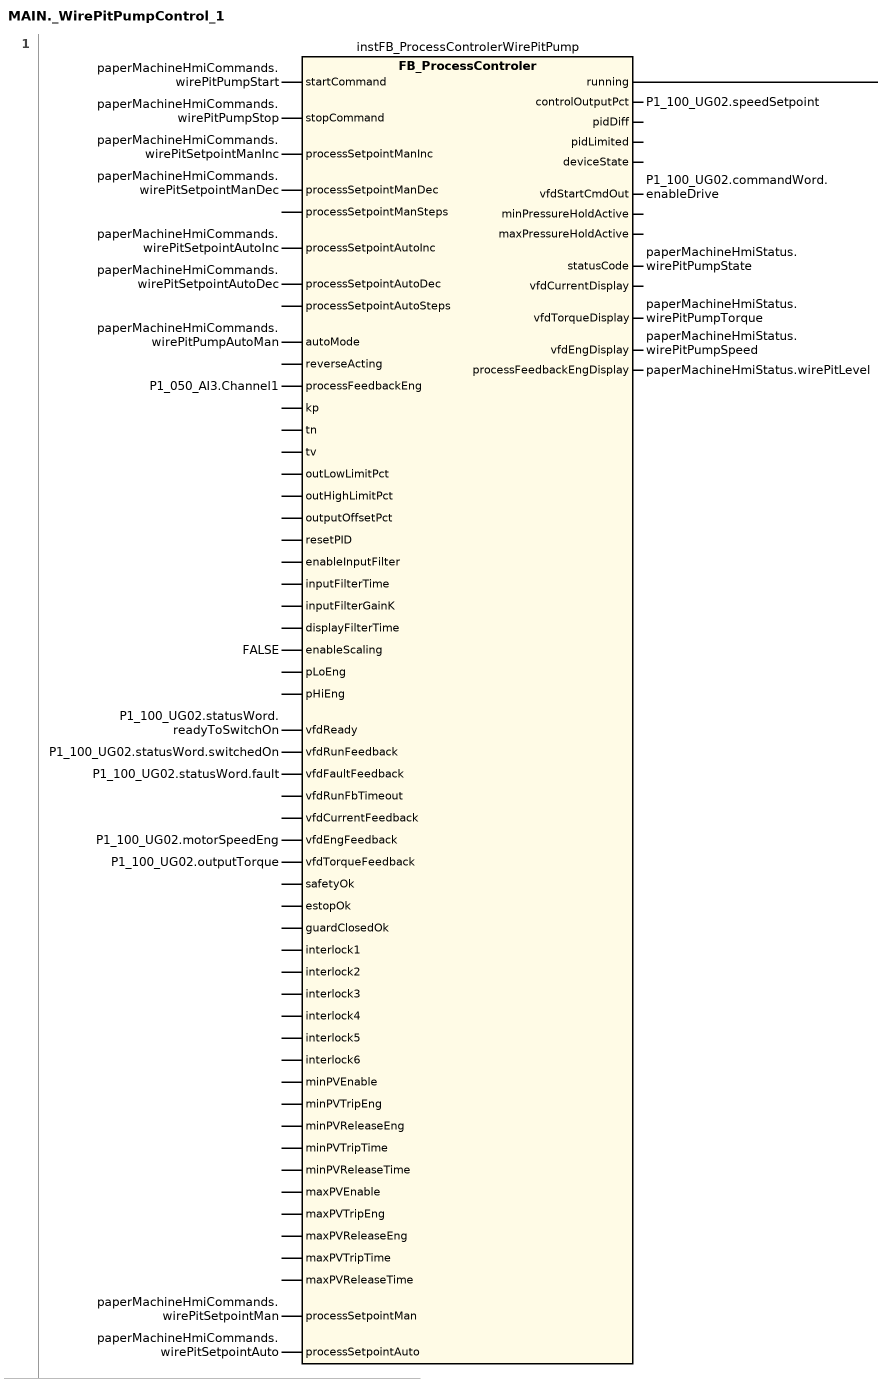
// NETWORK 1
instFB_ProcessControlerWirePitPump(
    startCommand := paperMachineHmiCommands.wirePitPumpStart,
    stopCommand := paperMachineHmiCommands.wirePitPumpStop,
    processSetpointManInc := paperMachineHmiCommands.wirePitSetpointManInc,
    processSetpointManDec := paperMachineHmiCommands.wirePitSetpointManDec,
    processSetpointAutoInc := paperMachineHmiCommands.wirePitSetpointAutoInc,
    processSetpointAutoDec := paperMachineHmiCommands.wirePitSetpointAutoDec,
    autoMode := paperMachineHmiCommands.wirePitPumpAutoMan,
    processFeedbackEng := P1_050_AI3.Channel1,
    enableScaling := FALSE,
    vfdReady := P1_100_UG02.statusWord.readyToSwitchOn,
    vfdRunFeedback := P1_100_UG02.statusWord.switchedOn,
    vfdFaultFeedback := P1_100_UG02.statusWord.fault,
    vfdEngFeedback := P1_100_UG02.motorSpeedEng,
    vfdTorqueFeedback := P1_100_UG02.outputTorque,
    processSetpointMan := paperMachineHmiCommands.wirePitSetpointMan,
    processSetpointAuto := paperMachineHmiCommands.wirePitSetpointAuto,
    controlOutputPct => P1_100_UG02.speedSetpoint,
    vfdStartCmdOut => P1_100_UG02.commandWord.enableDrive,
    statusCode => paperMachineHmiStatus.wirePitPumpState,
    vfdTorqueDisplay => paperMachineHmiStatus.wirePitPumpTorque,
    vfdEngDisplay => paperMachineHmiStatus.wirePitPumpSpeed,
    processFeedbackEngDisplay => paperMachineHmiStatus.wirePitLevel); // FB_ProcessControler
END_METHOD

METHOD machineReset
VAR_INPUT
END_VAR

VAR
	instTP_Reset: TP;
END_VAR
//────────────────────────────────────────────
// UG01 to UG06 (General Utilities / Aux Drives)
//────────────────────────────────────────────
P1_100_UG01.commandWord.faultResetCmd := paperMachineHmiCommands.machineReset;
P1_100_UG02.commandWord.faultResetCmd := paperMachineHmiCommands.machineReset;
P1_100_UG03_SuctionRoll.commandWord.faultResetCmd := paperMachineHmiCommands.machineReset;
P1_100_UG04.commandWord.faultResetCmd := paperMachineHmiCommands.machineReset;
P1_100_UG05.commandWord.faultResetCmd := paperMachineHmiCommands.machineReset;
P1_300_UG06_TractionRoll.commandWord.faultResetCmd := paperMachineHmiCommands.machineReset;

//────────────────────────────────────────────
// Safety PLC Reset
//────────────────────────────────────────────
P1_050_SP1.safetyReset := paperMachineHmiCommands.machineReset;
P1_050_SP1.errorAcknowledgement := paperMachineHmiCommands.machineReset;

//────────────────────────────────────────────
// Press Section Drives
//────────────────────────────────────────────
P11_400_UG01_SecondPress.commandWord.faultResetCmd := paperMachineHmiCommands.machineReset;
P12_400_UG01_FirstPress.commandWord.faultResetCmd := paperMachineHmiCommands.machineReset;

//────────────────────────────────────────────
// Drying Section — Group 1
//────────────────────────────────────────────
P13_500_UG01_1GR_UpperSlave.commandWord.faultResetCmd := paperMachineHmiCommands.machineReset;
P13_500_UG02_1GR_LowerMaster.commandWord.faultResetCmd := paperMachineHmiCommands.machineReset;
P13_500_UG03_1GR_UpperMaster.commandWord.faultResetCmd := paperMachineHmiCommands.machineReset;

//────────────────────────────────────────────
// Drying Section — Group 2
//────────────────────────────────────────────
P13_501_UG01_2GR_LowerSlave.commandWord.faultResetCmd := paperMachineHmiCommands.machineReset;
P13_501_UG02_2GR_UpperSlave.commandWord.faultResetCmd := paperMachineHmiCommands.machineReset;
P13_501_UG03_2GR_LowerMaster.commandWord.faultResetCmd := paperMachineHmiCommands.machineReset;
P14_501_UG01_2GR_UpperMaster.commandWord.faultResetCmd := paperMachineHmiCommands.machineReset;

//────────────────────────────────────────────
// Drying Section — Group 3
//────────────────────────────────────────────
P14_502_UG01_3GR_LowerSlave.commandWord.faultResetCmd := paperMachineHmiCommands.machineReset;
P14_502_UG02_3GR_UpperSlave.commandWord.faultResetCmd := paperMachineHmiCommands.machineReset;
P14_502_UG03_3GR_LowerMaster.commandWord.faultResetCmd := paperMachineHmiCommands.machineReset;
P14_502_UG04_3GR_UpperMaster.commandWord.faultResetCmd := paperMachineHmiCommands.machineReset;

//────────────────────────────────────────────
// Rewinder
//────────────────────────────────────────────
P15_600_UG01_Rewinder.commandWord.faultResetCmd := paperMachineHmiCommands.machineReset;
END_METHOD

END_PROGRAM

(* stored: Version 1.1.0.1, ProductVersion 3.1.4024.15
   POU MAIN: Id {5655f915-5dcf-4c87-91ff-2912e5ed07e4}, SpecialFunc None
   Method _000_Init_Variables: Id {5375a803-7613-4982-b9a2-f469ce258019}
   Method _001_FirstScan: Id {2b51631a-b1de-4251-88c9-0f83eb7f4089}
   Method _100_FormingBoardControl: Id {0c14a096-ab0f-45c1-953f-c1b000dd222b}
   Method _110_FormingBoardAux: Id {5aa4fd0c-47a3-4984-9a55-af92e2ae98ef}
   Method _200_PressSectionControl: Id {9f824a2c-9679-4031-8e2d-18b1073be726}
   Method _500_DryingSectionGroup1DriveControl: Id {7943a74e-10ea-458b-9502-2d49d50c4e35}
   Method _501_DryingSectionGroup2DriveControl: Id {f83f4d32-fa55-425e-9a54-fabf3c551fc1}
   Method _502_DryingSectionGroup3DriveControl: Id {9a974028-0ff1-4fc6-ae78-595db97cb730}
   Method _550_DryingSectionLubrification: Id {1c3ab415-b9c8-4039-a58e-5404ebefb0b7}
   Method _600_WinderGroup: Id {603ff0d1-31e4-4576-a200-a1a15c654d7f}
   Method _888_Alarms: Id {d9864b94-8b87-40be-9edc-0758f89dc5b9}
   Method _CentrifugalPressureScreenControl: Id {18b0f911-c9ca-4b47-826f-de0cd0c5db50}
   Method _CouchPitMixerControl: Id {98f7283d-3c51-4c62-91d0-f4e2606ab671}
   Method _CouchPitPumpControl: Id {60edba15-dfcb-4145-807a-b545f9976fa8}
   Method _FunctionBlockTest: Id {dc68dec4-b8e1-4e42-9c46-f76b6e3f7d02}
   Method _HeadBoxAuxiliaryControls: Id {b4d5fe16-43ef-431f-9e3b-d46cb5910730}
   Method _MixPumpControl_1: Id {d62a7ec7-6a8b-4696-bc00-270cd3d733f9}
   Method _StockPumpControl: Id {44ec4fcc-2a75-4e83-963c-b807cac52e25}
   Method _StockPumpControl_1: Id {f30519d5-f949-4cda-b919-d3c5e6fdcad4}
   Method _VaccumPumps: Id {8d03af37-1f90-4067-bf6c-04d0e3d98f21}
   Method _WirePitPumpControl: Id {b10dac86-1bc7-4eb2-913d-187a96879d44}
   Method _WirePitPumpControl_1: Id {7d4a518b-870d-4ab9-a21a-ca0bad9abb45}
   Method machineReset: Id {02d7d166-7912-45b0-ae8c-bd34367b2eb6} *)
